FUNCTION_BLOCK FB_MessageHandler
VAR_INPUT
END_VAR
VAR_OUTPUT
END_VAR
VAR
END_VAR

METHOD Report : BOOL
VAR_INPUT
END_VAR
END_METHOD

END_FUNCTION_BLOCK

(* stored: Version 1.1.0.1, ProductVersion 3.1.4024.10
   POU FB_MessageHandler: Id {5e483029-c47c-4224-84f9-f9b80035955b}, SpecialFunc None
   Method Report: Id {860efd01-b076-49c0-9779-74de16978f7d} *)
